FUNCTION_BLOCK Thermometer (* Service Interface Function Block Type *)
  (* Standard: 61499-1 Annex A; Description: Copyright (c) 2017 fortiss GmbH This program and the accompanying materials are made available under the terms of the Eclipse Public License 2.0 which is available at https://www.eclipse.org/legal/epl-2.0/ SPDX-License-Identifier: EPL-2.0 *)
  (* Version 1.0, 2017-09-21, Alois Zoitl, fortiss GmbH, initial API and implementation and/or initial documentation *)
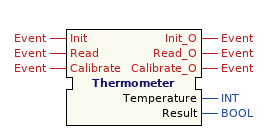
  EVENT_INPUT
    Init;
    Read;
    Calibrate;
  END_EVENT
  EVENT_OUTPUT
    Init_O;
    Read_O;
    Calibrate_O;
  END_EVENT
  VAR_OUTPUT
    Temperature : INT;
    Result : BOOL;
  END_VAR
END_FUNCTION_BLOCK
(* other elements stored in the file *)
(* SelfDiscription FBType=SENSOR *)
